// TIA Portal V19 export
DATA_BLOCK "Main_Safety_RTG1_DB"   // DB209, F_DB
AUTHOR : Siemens AG DI FA SUP
NAME : FUSI
// stored: InstanceOfName Safety.Main_Safety_RTG1, InstanceOfType FB, Namespace Safety
"Safety.Main_Safety_RTG1"
   // VAR
   //    status { ExternalAccessible := 'False'; ExternalVisible := 'False'; ExternalWritable := 'False'} : "Safety.typeDataFromSafety";
   //    statAck { ExternalWritable := 'False'} : Bool;
   //    instAckOP { ExternalWritable := 'False'} : ACK_OP;
   //    instAckGL { ExternalWritable := 'False'} : ACK_GL;
   //    instSafetyZone1Actuators { ExternalWritable := 'False'} : "Safety.SafetyZone1Actuators";
   //    instLSafeEStopDrvZone1 { ExternalWritable := 'False'} : "Safety.LSafe_EStopDrives";
   //    instLSafeFDoorDrvZone1 { ExternalWritable := 'False'} : "Safety.LSafe_FDoorDrives";
   //    instStatusSummary { ExternalWritable := 'False'} : "Safety.StatusSummary";
   // END_VAR
BEGIN
END_DATA_BLOCK
